FUNCTION_BLOCK FB_AlarmDiagnostic
VAR_INPUT
	i_bEnable				:BOOL:=TRUE;
	i_iID					:INT;
	i_bInput				:BOOL;
	i_iOnDelay				:DINT:=0;
	i_bReset				:BOOL;
	i_bTest					:BOOL;
	i_bActive				:BOOL;
	i_sDisplayText			:STRING:='';
END_VAR
VAR_OUTPUT
	q_bActive				:BOOL;
	q_iDetections			:INT;
END_VAR
VAR
	TON						:TON;
END_VAR
VAR // added by the converter: edge detectors and wires of the graphical bodies
    _rt1 : R_TRIG;
    _w1 : BOOL;
END_VAR

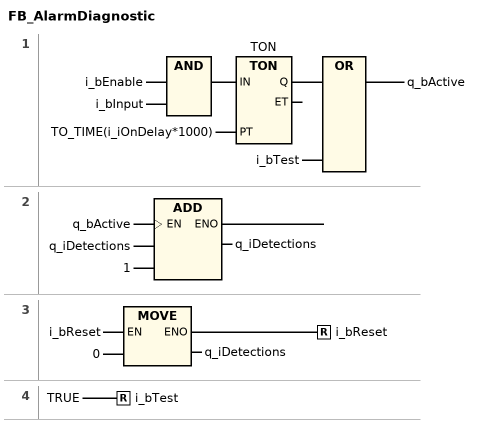
// NETWORK 1
TON(IN := i_bEnable AND i_bInput, PT := TO_TIME(i_iOnDelay*1000));
q_bActive := TON.Q OR i_bTest;

// NETWORK 2
_rt1(CLK := q_bActive);
IF _rt1.Q THEN q_iDetections := q_iDetections + 1; END_IF

// NETWORK 3
_w1 := i_bReset;
IF _w1 THEN q_iDetections := 0; END_IF
i_bReset R= _w1;

// NETWORK 4
i_bTest R= TRUE;

END_FUNCTION_BLOCK

(* stored: Version 1.1.0.1
   POU FB_AlarmDiagnostic: Id {f625d1c9-d47b-44f8-89f7-02fb4e944319}, SpecialFunc None *)
